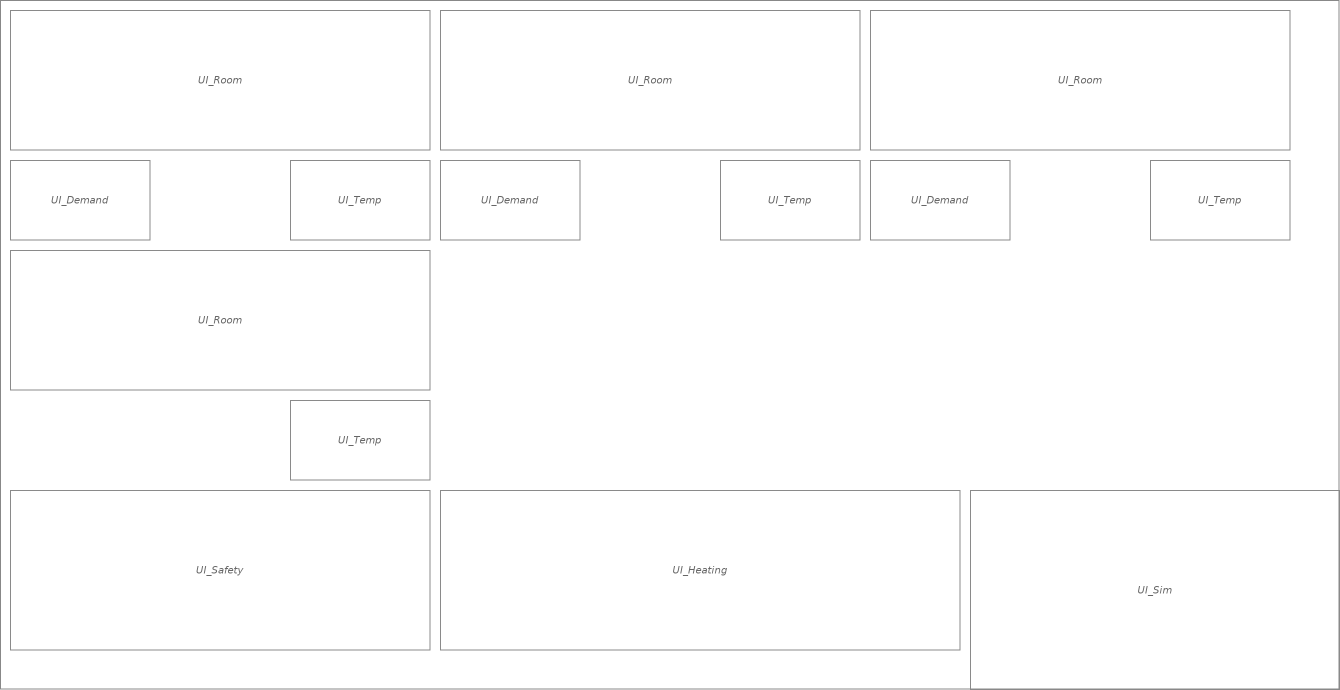
VISUALIZATION MAIN  // 1340x690
    Frame (10,490 420x160)
        shows UI_Safety(pou := MAIN.safety)
    Frame (440,490 520x160)
        shows UI_Heating(pou := MAIN.heating)
    Frame (970,490 370x200)
        shows UI_Sim(param := SIM.param)
    Frame (10,10 420x140)
        shows UI_Room(ctx := MAIN.stdRoom[1]._ctx)
    Frame (290,160 140x80)
        shows UI_Temp(hmi := MAIN.stdRoom[1]._lowTemperature._hmi)
    Frame (10,160 140x80)
        shows UI_Demand(hmi := MAIN.stdRoom[1]._demand._hmi)
    Frame (440,10 420x140)
        shows UI_Room(ctx := MAIN.stdRoom[2]._ctx)
    Frame (720,160 140x80)
        shows UI_Temp(hmi := MAIN.stdRoom[2]._lowTemperature._hmi)
    Frame (440,160 140x80)
        shows UI_Demand(hmi := MAIN.stdRoom[2]._demand._hmi)
    Frame (870,10 420x140)
        shows UI_Room(ctx := MAIN.stdRoom[3]._ctx)
    Frame (1150,160 140x80)
        shows UI_Temp(hmi := MAIN.stdRoom[3]._lowTemperature._hmi)
    Frame (870,160 140x80)
        shows UI_Demand(hmi := MAIN.stdRoom[3]._demand._hmi)
    Frame (10,250 420x140)
        shows UI_Room(ctx := MAIN.reception._ctx)
    Frame (290,400 140x80)
        shows UI_Temp(hmi := MAIN.reception._lowTemperature._hmi)
END_VISUALIZATION

(* stored: Version 1.1.0.1
   Visu MAIN: Id {1e026e4d-f1dc-41ee-aecc-8d5674db4a1b} *)
